PROGRAM MAIN
VAR
END_VAR

P_VCB();

END_PROGRAM

(* stored: Version 1.1.0.1, ProductVersion 3.1.4024.12
   POU MAIN: Id {ce645341-9c05-4cb3-833a-cdc75c30d821}, SpecialFunc None *)
